PROGRAM DAQTask
VAR
	EL3174			:MDP5001_300_B3F675AA;
	dataindex		:INT := 0;
	tempX			:INT;
	tempY			:INT;
	tempZ			:INT;
	prevX			:INT;
	prevY			:INT;
	prevZ			:INT;
	
	temptime		:ULINT;
	prevtime		:ULINT;	
	
    systemTime		:TIMESTRUCT;
	(*uses ADS functions that cannot guarantee real time execution*)
	fbTime			:FB_LocalSystemTime;
    timeAsDT		:DT;	
	timeASString	:STRING;	
	
	timer			:TON;
END_VAR

//1ms cycle time
fbTime(bEnable := TRUE, dwCycle := 1);
timeasstring := SYSTEMTIME_TO_STRING(fbtime.systemTime);
//calculate distance from massa sensor to surface (mm) and assign to temp variable
//out of range is represented by zero in temp variable
IF EL3174.MDP5001_300_Input.MDP5001_300_AI_Standard_Channel_1_Value = 0 THEN
	GVL_DAQ.DATA.MASSA_TEMP	:= 0;
ELSE
	GVL_DAQ.DATA.MASSA_TEMP	:= EL3174.MDP5001_300_Input.MDP5001_300_AI_Standard_Channel_1_Value * 2743/32767 + 101;
END_IF


//calculate distance from keyence sensor to sensor (mm) and assign to temp variable
//out of range is represented by zero in temp variable
//keyence set to high precision mode - 250mm to 450mm range.
//TODO measure range of motion for z axis
IF EL3174.MDP5001_300_Input.MDP5001_300_AI_Standard_Channel_2_Value = 32767 THEN
	GVL_DAQ.DATA.KEYENCE_TEMP 	:= 0;
ELSE
	GVL_DAQ.DATA.KEYENCE_TEMP	:= EL3174.MDP5001_300_Input.MDP5001_300_AI_Standard_Channel_2_Value * 100/32767 + 350;
END_IF


//TODO WriteData function is called in RunCommands based on selected sensors
//default acquire every mm - increase DAQINDEX decrease resolution
IF GVL_DAQ.DAQ_CTR_INT.Activate_Trigger <> DataTrigger.none THEN
	CASE GVL_DAQ.DAQ_CTR_INT.Activate_Trigger OF
		DataTrigger.none:;
		DataTrigger.x:
			tempX												:= LREAL_TO_INT(GVL_MOTION.xOut.PositionOut);
			IF tempX MOD GVL_DAQ.EXT_CTR.DAQACQRES = 0 AND (tempX <> prevX) THEN
				//timeASDT := SYSTEMTIME_TO_DT(fbtime.systemTime);
				GVL_DAQ.TIMESTAMP[GVL_DAQ.DATA_INDEX] 			:= DELETE(SYSTEMTIME_TO_STRING(fbtime.systemTime),11,1);

				GVL_DAQ.X[GVL_DAQ.DATA_INDEX] 			:= GVL_MOTION.xOut.PositionOut;
				GVL_DAQ.Y[GVL_DAQ.DATA_INDEX] 			:= GVL_MOTION.yOut.PositionOut;
				GVL_DAQ.Z[GVL_DAQ.DATA_INDEX] 			:= GVL_MOTION.zOut.PositionOut;
				
				GVL_DAQ.KEYENCE[GVL_DAQ.DATA_INDEX]		:= GVL_DAQ.DATA.KEYENCE_TEMP;
				GVL_DAQ.MASSA[GVL_DAQ.DATA_INDEX]		:= GVL_DAQ.DATA.MASSA_TEMP;
			
				
				GVL_DAQ.DATA_INDEX 								:= GVL_DAQ.DATA_INDEX + 1;
				IF (GVL_DAQ.DATA_INDEX >= 200000) THEN
					GVL_DAQ.DATA_INDEX 							:= 0;
					GVL_DAQ.DATA_OVERFLOW						:= TRUE;
				END_IF	
		
			END_IF	
			prevX												:= LREAL_TO_INT(GVL_MOTION.xOut.PositionOut);
		DataTrigger.y:
			tempY												:= LREAL_TO_INT(GVL_MOTION.yOut.PositionOut);
			IF tempY MOD GVL_DAQ.EXT_CTR.DAQACQRES = 0 AND (tempY <> prevY) THEN
				//timeASDT := SYSTEMTIME_TO_DT(fbtime.systemTime);
				GVL_DAQ.TIMESTAMP[GVL_DAQ.DATA_INDEX] 			:= DELETE(SYSTEMTIME_TO_STRING(fbtime.systemTime),11,1);
				
				GVL_DAQ.X[GVL_DAQ.DATA_INDEX] 			:= GVL_MOTION.xOut.PositionOut;
				GVL_DAQ.Y[GVL_DAQ.DATA_INDEX] 			:= GVL_MOTION.yOut.PositionOut;
				GVL_DAQ.Z[GVL_DAQ.DATA_INDEX] 			:= GVL_MOTION.zOut.PositionOut;
				
				GVL_DAQ.KEYENCE[GVL_DAQ.DATA_INDEX]		:= GVL_DAQ.DATA.KEYENCE_TEMP;
				GVL_DAQ.MASSA[GVL_DAQ.DATA_INDEX]		:= GVL_DAQ.DATA.MASSA_TEMP;
				
				GVL_DAQ.DATA_INDEX 								:= GVL_DAQ.DATA_INDEX + 1;
				IF (GVL_DAQ.DATA_INDEX >= 200000) THEN
					GVL_DAQ.DATA_INDEX 							:= 0;
					GVL_DAQ.DATA_OVERFLOW						:= TRUE;
				END_IF	
		
			END_IF
			prevY												:= LREAL_TO_INT(GVL_MOTION.yOut.PositionOut);
		DataTrigger.z:
			tempZ												:= LREAL_TO_INT(GVL_MOTION.zOut.PositionOut);
			IF tempZ MOD GVL_DAQ.EXT_CTR.DAQACQRES = 0 AND (tempZ <> prevZ) THEN
				//timeASDT := SYSTEMTIME_TO_DT(fbtime.systemTime);
				GVL_DAQ.TIMESTAMP[GVL_DAQ.DATA_INDEX] 			:= DELETE(SYSTEMTIME_TO_STRING(fbtime.systemTime),11,1);
					
				GVL_DAQ.X[GVL_DAQ.DATA_INDEX] 			:= GVL_MOTION.xOut.PositionOut;
				GVL_DAQ.Y[GVL_DAQ.DATA_INDEX] 			:= GVL_MOTION.yOut.PositionOut;
				GVL_DAQ.Z[GVL_DAQ.DATA_INDEX] 			:= GVL_MOTION.zOut.PositionOut;
				
				GVL_DAQ.KEYENCE[GVL_DAQ.DATA_INDEX]		:= GVL_DAQ.DATA.KEYENCE_TEMP;
				GVL_DAQ.MASSA[GVL_DAQ.DATA_INDEX]		:= GVL_DAQ.DATA.MASSA_TEMP;
				
				GVL_DAQ.DATA_INDEX 								:= GVL_DAQ.DATA_INDEX + 1;
				IF (GVL_DAQ.DATA_INDEX >= 200000) THEN
					GVL_DAQ.DATA_INDEX 							:= 0;
					GVL_DAQ.DATA_OVERFLOW						:= TRUE;
				END_IF	
		
			END_IF
			prevZ												:= LREAL_TO_INT(GVL_MOTION.zOut.PositionOut);
		DataTrigger.timed:
			temptime											:= F_GetSystemTime();
			IF ULINT_TO_LINT(temptime) MOD GVL_DAQ.EXT_CTR.DAQACQRES = 0 AND (temptime <> prevtime) THEN
				//timeASDT := SYSTEMTIME_TO_DT(fbtime.systemTime);
				GVL_DAQ.TIMESTAMP[GVL_DAQ.DATA_INDEX] 			:= DELETE(SYSTEMTIME_TO_STRING(fbtime.systemTime),11,1);
					
				GVL_DAQ.X[GVL_DAQ.DATA_INDEX] 			:= GVL_MOTION.xOut.PositionOut;
				GVL_DAQ.Y[GVL_DAQ.DATA_INDEX] 			:= GVL_MOTION.yOut.PositionOut;
				GVL_DAQ.Z[GVL_DAQ.DATA_INDEX] 			:= GVL_MOTION.zOut.PositionOut;
				
				GVL_DAQ.KEYENCE[GVL_DAQ.DATA_INDEX]		:= GVL_DAQ.DATA.KEYENCE_TEMP;
				GVL_DAQ.MASSA[GVL_DAQ.DATA_INDEX]		:= GVL_DAQ.DATA.MASSA_TEMP;
				
				GVL_DAQ.DATA_INDEX 								:= GVL_DAQ.DATA_INDEX + 1;
				IF (GVL_DAQ.DATA_INDEX >= 200000) THEN
					GVL_DAQ.DATA_INDEX 							:= 0;
					GVL_DAQ.DATA_OVERFLOW						:= TRUE;
				END_IF	
		
			END_IF			
			
			prevtime											:= F_GetSystemTime();
			
	END_CASE
ELSE
	tempX														:= 0;
	tempY														:= 0;
	tempZ														:= 0;
	prevX														:= 0;
	prevY														:= 0;
	prevZ														:= 0;		
END_IF

IF GVL_MOTION.EXT_CTR.AxesReset THEN
	GVL_DAQ.DAQ_CTR_INT.Activate_Trigger		:= DataTrigger.none;
END_IF

(*measure time taken for DAQ pass controlled by GVL_DAQ.DAQ_CTR_INT.Measure_Run_Time*)

DAQPassTime();

END_PROGRAM

(* stored: Version 1.1.0.1, ProductVersion 3.1.4026.12
   POU DAQTask: Id {82fb0ded-3f92-4d94-b129-9bf11d1d7a61}, SpecialFunc None *)
